FUNCTION_BLOCK CountFreeSpaces
VAR_INPUT
	DrinkArray: ARRAY [1..25] OF Drinks;
	PalletArray: ARRAY [1..25] OF BOOL;
END_VAR
VAR_OUTPUT
	FreeCola : INT;
	FreeFanta : INT;
END_VAR
VAR
	Counter : INT;
END_VAR

FreeCola := 0;
FreeFanta := 0;

FOR Counter:=1 TO 25 DO //sizeof array werkt niet
 	IF NOT PalletArray[Counter] THEN
		IF DrinkArray[Counter] = Drinks.Cola THEN
			FreeCola:= FreeCola + 1;
		ELSE
			FreeFanta:= FreeFanta + 1;
		END_IF
	END_IF
END_FOR

END_FUNCTION_BLOCK

(* stored: Version 1.1.0.1, ProductVersion 3.1.4022.12
   POU CountFreeSpaces: Id {582a3d25-c141-4dd7-ac3d-738e01933621}, SpecialFunc None *)
